(* IEC 61131-3 sources: s32-hmi/, 2 files *)

(* ---- state-machine.st ---- *)
(*
===============================================================================
VOLTAGRID / SEL RTAC MASTER CONTROLLER
STATE-MACHINE SKELETON
Single Master Controller Version
-------------------------------------------------------------------------------
Intent:
- Supervisory coordination only
- Local genset controllers, SEL relays, SEL-2240, OEM controllers retain
  machine/protection ownership
- Master issues permissives, start/stop requests, breaker open/close requests,
  AGC/VCS biases, and orchestrates major sequences
===============================================================================
*)

(*
===============================================================================
TYPE DECLARATIONS
===============================================================================
*)
TYPE E_SYS_STATE :
(
    SYS_INIT := 0,
    SYS_IDLE := 1,
    SYS_NORMAL := 2,
    SYS_PARTY_MODE := 3,
    SYS_BLACKOUT_DETECTED := 4,
    SYS_BLACKOUT_RECOVERY := 5,
    SYS_BLACKSTART_READY := 6,
    SYS_BLACKSTART_ACTIVE := 7,
    SYS_FAULT := 8,
    SYS_ABORTED := 9
);
END_TYPE

TYPE E_SEQ_STATE :
(
    SEQ_IDLE := 0,
    SEQ_START := 1,
    SEQ_CHECK_PERMISSIVES := 2,
    SEQ_ISSUE_COMMAND := 3,
    SEQ_WAIT_FEEDBACK := 4,
    SEQ_VERIFY := 5,
    SEQ_COMPLETE := 6,
    SEQ_FAIL := 7,
    SEQ_ABORT := 8
);
END_TYPE

TYPE E_GEN_MODE :
(
    GEN_BLOCK := 0,
    GEN_STOP := 1,
    GEN_AUTO := 2,
    GEN_MANUAL := 3
);
END_TYPE

TYPE E_GEN_RUN_STATE :
(
    GEN_OFFLINE := 0,
    GEN_STARTING := 1,
    GEN_RUNNING_UNSYNC := 2,
    GEN_SYNCED := 3,
    GEN_STOPPING := 4,
    GEN_TRIPPED := 5,
    GEN_UNAVAILABLE := 6
);
END_TYPE

TYPE E_BREAKER_STATE :
(
    BRK_OPEN := 0,
    BRK_CLOSED := 1,
    BRK_TRANSITION := 2,
    BRK_FAIL := 3,
    BRK_UNKNOWN := 4
);
END_TYPE

TYPE ST_Genset :
STRUCT
    Id                      : INT;
    Enabled                 : BOOL;
    ModeCmd                 : E_GEN_MODE;     (* from HMI *)
    Priority                : INT;            (* 1..100 *)
    EngineHours             : REAL;

    (* permissives / feedback *)
    LocalReadyForDemand     : BOOL;           (* DIA.NE / OEM / Modbus *)
    InAutoAtLocal           : BOOL;
    NoStartBlockAlarms      : BOOL;
    RunningFb               : BOOL;
    SyncCompleteFb          : BOOL;
    GCB_ClosedFb            : BOOL;
    TripFb                  : BOOL;
    DelayedShutdownReqFb    : BOOL;

    (* measured *)
    kW                      : REAL;
    kVAR                    : REAL;
    AvailablekW             : REAL;

    (* supervisory outputs *)
    StartReq                : BOOL;
    StopReq                 : BOOL;
    RemoteBlockCmd          : BOOL;
    PlantEmergencyModeCmd   : BOOL;
    FastDisconnectCmd       : BOOL;
    FullThrottleModeCmd     : BOOL;

    AGC_Enable              : BOOL;
    AGC_Manual              : BOOL;
    AGC_kW_Setpoint         : REAL;
    AGC_kW_Min              : REAL;
    AGC_kW_Max              : REAL;
    AGC_BiasOut             : REAL;           (* abstract bias output *)

    VCS_Enable              : BOOL;
    VCS_Manual              : BOOL;
    VCS_kVAR_Setpoint       : REAL;
    VCS_kVAR_Min            : REAL;
    VCS_kVAR_Max            : REAL;
    VCS_BiasOut             : REAL;           (* abstract bias output *)

    RunState                : E_GEN_RUN_STATE;
    StartPermissive         : BOOL;
    StopPermissive          : BOOL;
    SelectedForStart        : BOOL;
    SelectedForStop         : BOOL;
END_STRUCT
END_TYPE

TYPE ST_Breaker :
STRUCT
    Id                      : INT;
    Name                    : STRING[40];
    ControlEnabled          : BOOL;
    RatedAmps               : INT;

    OpenFb                  : BOOL;
    ClosedFb                : BOOL;
    TripAlarmFb             : BOOL;
    BusVoltage              : REAL;

    OpenCmd                 : BOOL;
    CloseCmd                : BOOL;
    BlockClose              : BOOL;

    State                   : E_BREAKER_STATE;
    SeqState                : E_SEQ_STATE;
END_STRUCT
END_TYPE

TYPE ST_System :
STRUCT
    State                   : E_SYS_STATE;
    PrevState               : E_SYS_STATE;

    HealthyMaster           : BOOL;
    HealthyComms            : BOOL;
    HMI_HeartbeatOk         : BOOL;
    OT_Healthy              : BOOL;

    PartyModeReq            : BOOL;
    PartyModeActive         : BOOL;
    BlackStartEnable        : BOOL;
    BlackStartReq           : BOOL;
    BlackStartActive        : BOOL;

    BlackoutDetected        : BOOL;
    DeadBus34k5             : BOOL;
    DeadBus480              : BOOL;

    IRM_TargetPct           : REAL;
    MinimumSynchronized     : INT;
    MinGensetLoadPct        : REAL;

    Plant_kW_Load           : REAL;
    Plant_kVAR              : REAL;
    MainBus_kV              : REAL;
    MainBus_Hz              : REAL;

    AlarmActive             : BOOL;
    FaultLatched            : BOOL;
    AbortReq                : BOOL;
    ResetReq                : BOOL;
END_STRUCT
END_TYPE

(*
===============================================================================
GLOBAL VARIABLES
===============================================================================
*)
VAR_GLOBAL
    gSys            : ST_System;
    gGensets        : ARRAY[1..46] OF ST_Genset;      (* size adapt per site *)
    gMVBreakers     : ARRAY[1..200] OF ST_Breaker;    (* site-specific *)
    gLVBreakers     : ARRAY[1..200] OF ST_Breaker;    (* site-specific *)
END_VAR

(*
===============================================================================
UTILITY FUNCTIONS
===============================================================================
*)
FUNCTION F_IsDeadBus : BOOL
VAR_INPUT
    Bus_kV          : REAL;
    Nominal_kV      : REAL;
    ThresholdPU     : REAL;       (* e.g. 0.3 *)
END_VAR
F_IsDeadBus := (Bus_kV < (Nominal_kV * ThresholdPU));

FUNCTION F_GensetStartPermissive : BOOL
VAR_INPUT
    Gen             : ST_Genset;
END_VAR
F_GensetStartPermissive :=
    Gen.Enabled
    AND (Gen.ModeCmd = GEN_AUTO)
    AND Gen.LocalReadyForDemand
    AND Gen.InAutoAtLocal
    AND Gen.NoStartBlockAlarms
    AND NOT Gen.TripFb;

FUNCTION F_GensetStopPermissive : BOOL
VAR_INPUT
    Gen             : ST_Genset;
END_VAR
F_GensetStopPermissive :=
    Gen.Enabled
    AND (Gen.RunState = GEN_SYNCED OR Gen.RunState = GEN_RUNNING_UNSYNC)
    AND NOT Gen.TripFb;

FUNCTION F_AverageOnlineLoadPct : REAL
VAR
    i               : INT;
    n               : INT;
    totalPct        : REAL;
    pct             : REAL;
END_VAR
n := 0;
totalPct := 0.0;

FOR i := 1 TO 46 DO
    IF gGensets[i].RunState = GEN_SYNCED THEN
        IF gGensets[i].AvailablekW > 0.0 THEN
            pct := (gGensets[i].kW / gGensets[i].AvailablekW) * 100.0;
            totalPct := totalPct + pct;
            n := n + 1;
        END_IF;
    END_IF;
END_FOR;

IF n > 0 THEN
    F_AverageOnlineLoadPct := totalPct / INT_TO_REAL(n);
ELSE
    F_AverageOnlineLoadPct := 0.0;
END_IF;

FUNCTION F_OnlineGenCount : INT
VAR
    i               : INT;
    n               : INT;
END_VAR
n := 0;
FOR i := 1 TO 46 DO
    IF gGensets[i].RunState = GEN_SYNCED THEN
        n := n + 1;
    END_IF;
END_FOR;
F_OnlineGenCount := n;

FUNCTION F_RequiredGenCountIRM : INT
VAR_INPUT
    PlantLoadkW         : REAL;
    IRM_TargetPct       : REAL;
END_VAR
VAR
    RequiredCapacity    : REAL;
    i                   : INT;
    sortedCap           : ARRAY[1..46] OF REAL;
    sumCap              : REAL;
    cnt                 : INT;
END_VAR

(* Skeleton only:
   Required online count = enough online available kW so that
   reserve margin >= IRM_TargetPct.
*)
RequiredCapacity := PlantLoadkW * (1.0 + (IRM_TargetPct / 100.0));
sumCap := 0.0;
cnt := 0;

FOR i := 1 TO 46 DO
    IF gGensets[i].Enabled THEN
        cnt := cnt + 1;
        sortedCap[cnt] := gGensets[i].AvailablekW;
    END_IF;
END_FOR;

(* TODO: sort by commitment preference / priority class *)
sumCap := 0.0;
F_RequiredGenCountIRM := 0;
FOR i := 1 TO cnt DO
    sumCap := sumCap + sortedCap[i];
    F_RequiredGenCountIRM := F_RequiredGenCountIRM + 1;
    IF sumCap >= RequiredCapacity THEN
        EXIT;
    END_IF;
END_FOR;

(*
===============================================================================
FUNCTION BLOCKS
===============================================================================
*)
FUNCTION_BLOCK FB_GensetState
VAR_INPUT
    Id              : INT;
END_VAR
VAR
    StartPerm       : BOOL;
    StopPerm        : BOOL;
END_VAR

StartPerm := F_GensetStartPermissive(Gen := gGensets[Id]);
StopPerm  := F_GensetStopPermissive(Gen := gGensets[Id]);

gGensets[Id].StartPermissive := StartPerm;
gGensets[Id].StopPermissive  := StopPerm;

IF gGensets[Id].TripFb THEN
    gGensets[Id].RunState := GEN_TRIPPED;

ELSIF gGensets[Id].RunningFb AND gGensets[Id].GCB_ClosedFb AND gGensets[Id].SyncCompleteFb THEN
    gGensets[Id].RunState := GEN_SYNCED;

ELSIF gGensets[Id].RunningFb AND NOT gGensets[Id].GCB_ClosedFb THEN
    gGensets[Id].RunState := GEN_RUNNING_UNSYNC;

ELSIF gGensets[Id].StartReq AND NOT gGensets[Id].RunningFb THEN
    gGensets[Id].RunState := GEN_STARTING;

ELSIF gGensets[Id].StopReq AND gGensets[Id].RunningFb THEN
    gGensets[Id].RunState := GEN_STOPPING;

ELSIF NOT gGensets[Id].RunningFb THEN
    gGensets[Id].RunState := GEN_OFFLINE;

ELSE
    (* hold last *)
END_IF;

FUNCTION_BLOCK FB_AGC_VCS
VAR
    i               : INT;
    OnlineCount     : INT;
    HzError         : REAL;
    kVError         : REAL;
    SharedkWBias    : REAL;
    SharedkVARBias  : REAL;
END_VAR

OnlineCount := F_OnlineGenCount();

(* Skeleton only *)
HzError := 60.0 - gSys.MainBus_Hz;
kVError := 34.5 - gSys.MainBus_kV;

SharedkWBias := HzError * 100.0;
SharedkVARBias := kVError * 100.0;

FOR i := 1 TO 46 DO
    IF gGensets[i].RunState = GEN_SYNCED THEN

        IF gGensets[i].AGC_Enable THEN
            IF gGensets[i].AGC_Manual THEN
                gGensets[i].AGC_BiasOut := gGensets[i].AGC_kW_Setpoint;
            ELSE
                gGensets[i].AGC_BiasOut := SharedkWBias / INT_TO_REAL(MAX(OnlineCount,1));
            END_IF;
        ELSE
            gGensets[i].AGC_BiasOut := 0.0;
        END_IF;

        IF gGensets[i].VCS_Enable THEN
            IF gGensets[i].VCS_Manual THEN
                gGensets[i].VCS_BiasOut := gGensets[i].VCS_kVAR_Setpoint;
            ELSE
                gGensets[i].VCS_BiasOut := SharedkVARBias / INT_TO_REAL(MAX(OnlineCount,1));
            END_IF;
        ELSE
            gGensets[i].VCS_BiasOut := 0.0;
        END_IF;

        (* clamp *)
        IF gGensets[i].AGC_BiasOut < gGensets[i].AGC_kW_Min THEN
            gGensets[i].AGC_BiasOut := gGensets[i].AGC_kW_Min;
        END_IF;
        IF gGensets[i].AGC_BiasOut > gGensets[i].AGC_kW_Max THEN
            gGensets[i].AGC_BiasOut := gGensets[i].AGC_kW_Max;
        END_IF;

        IF gGensets[i].VCS_BiasOut < gGensets[i].VCS_kVAR_Min THEN
            gGensets[i].VCS_BiasOut := gGensets[i].VCS_kVAR_Min;
        END_IF;
        IF gGensets[i].VCS_BiasOut > gGensets[i].VCS_kVAR_Max THEN
            gGensets[i].VCS_BiasOut := gGensets[i].VCS_kVAR_Max;
        END_IF;
    ELSE
        gGensets[i].AGC_BiasOut := 0.0;
        gGensets[i].VCS_BiasOut := 0.0;
    END_IF;
END_FOR;

FUNCTION_BLOCK FB_GMS
VAR
    i                   : INT;
    OnlineCount         : INT;
    RequiredCount       : INT;
    AvgLoadPct          : REAL;
    StartIssued         : INT;
    StopCandidate       : INT;
END_VAR

OnlineCount := F_OnlineGenCount();
RequiredCount := F_RequiredGenCountIRM(
                    PlantLoadkW := gSys.Plant_kW_Load,
                    IRM_TargetPct := gSys.IRM_TargetPct);
IF RequiredCount < gSys.MinimumSynchronized THEN
    RequiredCount := gSys.MinimumSynchronized;
END_IF;

AvgLoadPct := F_AverageOnlineLoadPct();

(* clear selections *)
FOR i := 1 TO 46 DO
    gGensets[i].SelectedForStart := FALSE;
    gGensets[i].SelectedForStop := FALSE;
END_FOR;

(* Party Mode bypasses automatic GMS *)
IF gSys.PartyModeActive THEN
    RETURN;
END_IF;

(* Start logic: IRM has priority *)
IF OnlineCount < RequiredCount THEN
    StartIssued := 0;

    (* Skeleton selection:
       Choose two startable gensets by best priority / least hours tie-break
    *)
    FOR i := 1 TO 46 DO
        IF F_GensetStartPermissive(Gen := gGensets[i]) AND (gGensets[i].RunState = GEN_OFFLINE) THEN
            gGensets[i].SelectedForStart := TRUE;
            gGensets[i].StartReq := TRUE;
            StartIssued := StartIssued + 1;
        END_IF;

        IF StartIssued >= 2 THEN
            EXIT;
        END_IF;
    END_FOR;
END_IF;

(* Stop logic: only if above IRM need and minimum load violated *)
IF (OnlineCount > RequiredCount) AND (AvgLoadPct < gSys.MinGensetLoadPct) THEN
    StopCandidate := 0;

    (* Skeleton selection:
       Highest engine hours among equal priorities, lowest commitment value first
    *)
    FOR i := 1 TO 46 DO
        IF F_GensetStopPermissive(Gen := gGensets[i]) THEN
            StopCandidate := i;
            EXIT;
        END_IF;
    END_FOR;

    IF StopCandidate > 0 THEN
        gGensets[StopCandidate].SelectedForStop := TRUE;
        gGensets[StopCandidate].StopReq := TRUE;
    END_IF;
END_IF;

(* delayed shutdown override *)
FOR i := 1 TO 46 DO
    IF gGensets[i].DelayedShutdownReqFb THEN
        (* maintain IRM by demanding extra gensets *)
        (* skeleton: flag handled naturally by RequiredCount/start logic *)
    END_IF;
END_FOR;

FUNCTION_BLOCK FB_PartyMode
VAR
    i               : INT;
END_VAR

gSys.PartyModeActive := gSys.PartyModeReq;

IF gSys.PartyModeActive THEN
    FOR i := 1 TO 46 DO
        IF F_GensetStartPermissive(Gen := gGensets[i]) THEN
            gGensets[i].StartReq := TRUE;
        END_IF;
    END_FOR;
END_IF;

FUNCTION_BLOCK FB_BlackoutRecovery
VAR
    Seq             : E_SEQ_STATE := SEQ_IDLE;
    TimerExpired    : BOOL;
    i               : INT;
END_VAR

CASE Seq OF

SEQ_IDLE:
    IF gSys.BlackoutDetected THEN
        Seq := SEQ_START;
    END_IF;

SEQ_START:
    (* Verify master and comms healthy *)
    IF gSys.HealthyMaster AND gSys.HealthyComms THEN
        Seq := SEQ_CHECK_PERMISSIVES;
    ELSE
        Seq := SEQ_FAIL;
    END_IF;

SEQ_CHECK_PERMISSIVES:
    gSys.DeadBus34k5 := F_IsDeadBus(Bus_kV := gSys.MainBus_kV, Nominal_kV := 34.5, ThresholdPU := 0.3);
    (* gSys.DeadBus480 to come from LV E-house measurement *)
    IF gSys.DeadBus34k5 AND gSys.DeadBus480 THEN
        Seq := SEQ_ISSUE_COMMAND;
    END_IF;

SEQ_ISSUE_COMMAND:
    (* Open all ICBs + LV feeders required by site logic *)
    FOR i := 1 TO 200 DO
        IF gMVBreakers[i].ControlEnabled THEN
            gMVBreakers[i].OpenCmd := TRUE;
        END_IF;
        IF gLVBreakers[i].ControlEnabled THEN
            gLVBreakers[i].OpenCmd := TRUE;
        END_IF;
    END_FOR;

    (* Start backup diesel through OEM controller / EMCP interface *)
    (* BackupDiesel.StartReq := TRUE; *)
    Seq := SEQ_WAIT_FEEDBACK;

SEQ_WAIT_FEEDBACK:
    (* wait for breaker feedback and backup diesel online *)
    (* skeleton: replace with timers and feedback checks *)
    TimerExpired := FALSE;
    IF NOT TimerExpired THEN
        Seq := SEQ_VERIFY;
    ELSE
        Seq := SEQ_FAIL;
    END_IF;

SEQ_VERIFY:
    (* close critical LV feeders only *)
    (* issue site-specific close list *)
    Seq := SEQ_COMPLETE;

SEQ_COMPLETE:
    gSys.State := SYS_BLACKSTART_READY;
    (* hold complete *)

SEQ_FAIL:
    gSys.AlarmActive := TRUE;
    gSys.FaultLatched := TRUE;
    IF gSys.AbortReq THEN
        Seq := SEQ_ABORT;
    ELSIF gSys.ResetReq THEN
        Seq := SEQ_IDLE;
    END_IF;

SEQ_ABORT:
    gSys.State := SYS_ABORTED;

END_CASE;

FUNCTION_BLOCK FB_BlackStart
VAR
    Seq             : E_SEQ_STATE := SEQ_IDLE;
    i               : INT;
    StartedPrimary  : INT;
END_VAR

CASE Seq OF

SEQ_IDLE:
    IF gSys.BlackStartReq AND gSys.BlackStartEnable AND (gSys.State = SYS_BLACKSTART_READY) THEN
        Seq := SEQ_START;
    END_IF;

SEQ_START:
    gSys.BlackStartActive := TRUE;
    Seq := SEQ_CHECK_PERMISSIVES;

SEQ_CHECK_PERMISSIVES:
    IF gSys.HealthyMaster AND gSys.HealthyComms AND gSys.DeadBus34k5 THEN
        Seq := SEQ_ISSUE_COMMAND;
    ELSE
        Seq := SEQ_FAIL;
    END_IF;

SEQ_ISSUE_COMMAND:
    (* example sequence:
       1) verify all ICBs open
       2) close SYNCON path if required
       3) energize main bus
       4) start/stage gensets
       5) transfer off backup diesel
    *)

    (* step: start two primary gensets *)
    StartedPrimary := 0;
    FOR i := 1 TO 46 DO
        IF F_GensetStartPermissive(Gen := gGensets[i]) THEN
            gGensets[i].StartReq := TRUE;
            StartedPrimary := StartedPrimary + 1;
        END_IF;

        IF StartedPrimary >= 2 THEN
            EXIT;
        END_IF;
    END_FOR;

    Seq := SEQ_WAIT_FEEDBACK;

SEQ_WAIT_FEEDBACK:
    (* wait for running/sync feedback *)
    Seq := SEQ_VERIFY;

SEQ_VERIFY:
    (* if enough primary gensets synced, isolate backup diesel *)
    IF F_OnlineGenCount() >= gSys.MinimumSynchronized THEN
        (* BackupDiesel.StopReq := TRUE; *)
        gSys.BlackStartActive := FALSE;
        Seq := SEQ_COMPLETE;
    ELSE
        Seq := SEQ_FAIL;
    END_IF;

SEQ_COMPLETE:
    gSys.State := SYS_NORMAL;

SEQ_FAIL:
    gSys.AlarmActive := TRUE;
    gSys.FaultLatched := TRUE;
    IF gSys.AbortReq THEN
        Seq := SEQ_ABORT;
    ELSIF gSys.ResetReq THEN
        Seq := SEQ_IDLE;
    END_IF;

SEQ_ABORT:
    gSys.BlackStartActive := FALSE;
    gSys.State := SYS_ABORTED;

END_CASE;

FUNCTION_BLOCK FB_BreakerState
VAR_INPUT
    IsLV            : BOOL;
    Id              : INT;
END_VAR

IF IsLV THEN
    IF gLVBreakers[Id].OpenFb AND NOT gLVBreakers[Id].ClosedFb THEN
        gLVBreakers[Id].State := BRK_OPEN;
    ELSIF gLVBreakers[Id].ClosedFb AND NOT gLVBreakers[Id].OpenFb THEN
        gLVBreakers[Id].State := BRK_CLOSED;
    ELSIF gLVBreakers[Id].TripAlarmFb THEN
        gLVBreakers[Id].State := BRK_FAIL;
    ELSE
        gLVBreakers[Id].State := BRK_UNKNOWN;
    END_IF;
ELSE
    IF gMVBreakers[Id].OpenFb AND NOT gMVBreakers[Id].ClosedFb THEN
        gMVBreakers[Id].State := BRK_OPEN;
    ELSIF gMVBreakers[Id].ClosedFb AND NOT gMVBreakers[Id].OpenFb THEN
        gMVBreakers[Id].State := BRK_CLOSED;
    ELSIF gMVBreakers[Id].TripAlarmFb THEN
        gMVBreakers[Id].State := BRK_FAIL;
    ELSE
        gMVBreakers[Id].State := BRK_UNKNOWN;
    END_IF;
END_IF;

(*
===============================================================================
PROGRAMS
===============================================================================
*)
PROGRAM PRG_InputMapping
VAR
    i               : INT;
END_VAR

(* Map site I/O, FEP tags, relay bits, SEL-2411 data, Modbus data here *)

FOR i := 1 TO 46 DO
    (* Example abstractions only:
       gGensets[i].LocalReadyForDemand := <from SEL-2411 hardwire or Modbus>;
       gGensets[i].RunningFb := <from SEL-2411 or OEM>;
       gGensets[i].GCB_ClosedFb := <from SEL-700G>;
       gGensets[i].SyncCompleteFb := <from OEM / relay>;
       gGensets[i].TripFb := <from OEM/relay>;
       gGensets[i].kW := <analog>;
       gGensets[i].kVAR := <analog>;
       gGensets[i].AvailablekW := <analog>;
       gGensets[i].EngineHours := <Modbus>;
    *)
END_FOR;

(* example Holt-style mapping candidate *)
(*
   Engine Start/Stop write reg: 0x006C
   Engine operating mode read: 0x0000 / 0x00A2
   Starter mode read: 0x021A
   Start-stop state read: 0x009A
   Shutdown active alarm: 0x0281
*)

PROGRAM PRG_SupervisoryState
VAR
    blackoutFB      : FB_BlackoutRecovery;
    blackstartFB    : FB_BlackStart;
END_VAR

gSys.DeadBus34k5 := F_IsDeadBus(Bus_kV := gSys.MainBus_kV, Nominal_kV := 34.5, ThresholdPU := 0.3);

CASE gSys.State OF

SYS_INIT:
    IF gSys.HealthyMaster THEN
        gSys.State := SYS_IDLE;
    END_IF;

SYS_IDLE:
    IF gSys.BlackoutDetected THEN
        gSys.State := SYS_BLACKOUT_DETECTED;
    ELSE
        gSys.State := SYS_NORMAL;
    END_IF;

SYS_NORMAL:
    IF gSys.PartyModeReq THEN
        gSys.State := SYS_PARTY_MODE;
    ELSIF gSys.BlackoutDetected THEN
        gSys.State := SYS_BLACKOUT_DETECTED;
    ELSIF gSys.FaultLatched THEN
        gSys.State := SYS_FAULT;
    END_IF;

SYS_PARTY_MODE:
    IF NOT gSys.PartyModeReq THEN
        gSys.State := SYS_NORMAL;
    END_IF;

SYS_BLACKOUT_DETECTED:
    gSys.State := SYS_BLACKOUT_RECOVERY;

SYS_BLACKOUT_RECOVERY:
    blackoutFB();
    IF gSys.State = SYS_BLACKSTART_READY THEN
        (* transition done in FB *)
    END_IF;

SYS_BLACKSTART_READY:
    IF gSys.BlackStartReq THEN
        gSys.State := SYS_BLACKSTART_ACTIVE;
    END_IF;

SYS_BLACKSTART_ACTIVE:
    blackstartFB();

SYS_FAULT:
    IF gSys.ResetReq THEN
        gSys.FaultLatched := FALSE;
        gSys.State := SYS_IDLE;
    END_IF;

SYS_ABORTED:
    IF gSys.ResetReq THEN
        gSys.State := SYS_IDLE;
    END_IF;

END_CASE;

PROGRAM PRG_GeneratorSupervisor
VAR
    i               : INT;
    genFB           : ARRAY[1..46] OF FB_GensetState;
    agcFB           : FB_AGC_VCS;
    gmsFB           : FB_GMS;
    partyFB         : FB_PartyMode;
END_VAR

FOR i := 1 TO 46 DO
    genFB[i](Id := i);
END_FOR;

partyFB();

IF (gSys.State = SYS_NORMAL) OR (gSys.State = SYS_PARTY_MODE) THEN
    gmsFB();
    agcFB();
END_IF;

PROGRAM PRG_BreakerSupervisor
VAR
    i               : INT;
    mvFB            : ARRAY[1..200] OF FB_BreakerState;
    lvFB            : ARRAY[1..200] OF FB_BreakerState;
END_VAR

FOR i := 1 TO 200 DO
    mvFB[i](IsLV := FALSE, Id := i);
    lvFB[i](IsLV := TRUE, Id := i);
END_FOR;

PROGRAM PRG_OutputMapping
VAR
    i               : INT;
END_VAR

FOR i := 1 TO 46 DO
    (* map supervisory requests to real outputs / comm writes *)

    (* hardwire style *)
    (*
    SEL2411_OUT_Start[i] := PulseFromBool(gGensets[i].StartReq);
    SEL2411_OUT_Stop[i] := PulseFromBool(gGensets[i].StopReq);
    SEL2411_OUT_RemoteBlock[i] := gGensets[i].RemoteBlockCmd;
    SEL2411_AO_kWSetpoint[i] := gGensets[i].AGC_BiasOut;
    SEL2411_AO_kVARSetpoint[i] := gGensets[i].VCS_BiasOut;
    *)

    (* Modbus style alternative *)
    (*
    IF gGensets[i].StartReq THEN
        ModbusWrite(Reg := 16#006C, Value := 2);   (* RUN *)
    ELSIF gGensets[i].StopReq THEN
        ModbusWrite(Reg := 16#006C, Value := 0);   (* STOP *)
    END_IF;
    *)
END_FOR;

FOR i := 1 TO 200 DO
    (* map MV and LV breaker commands to FEP/relay/2240 interface *)
    (* NGVL -> FEP -> GOOSE/MMS/Modbus *)
END_FOR;

PROGRAM PLC_PRG
PRG_InputMapping();
PRG_SupervisoryState();
PRG_GeneratorSupervisor();
PRG_BreakerSupervisor();
PRG_OutputMapping();

(* ---- load-bank-main.st ---- *)
PROGRAM Main_Main_Man
VAR
	Test_Run : BOOL;

	Burn_In : TON;
	Current_Burn_In_Time : TIME;

	Load_Bank_Gateway_Software_Version : DINT;
	Load_Bank_Load_Accept_Sync : DINT;
	Load_Bank_Load_Accept_Reject : DINT;
	Load_Bank_Load_Bank_Count : DINT;
	Load_Bank_Nominal_Voltage : DINT;
	Load_Bank_Nominal_Frequency : DINT;
	Load_Bank_Connection_Mode : DINT;
	Load_Bank_Min_Resistive_Load_Step : UDINT;
	Load_Bank_Measured_Active_Power : DINT;
	Load_Bank_Applied_Resistive_Load : UDINT;
	Load_Bank_Requested_Resistive_Load : UDINT;
	Load_Bank_Requested_Resistive_Load_2 : UDINT;
	Load_Bank_Network_Rescan : DINT;
	Load_Bank_System_Status : DINT;
	Load_Bank_System_Alarms : DINT;
	Load_Bank_Available_Resistive_Load : UDINT;
	Test_Value : DINT;

	Gen_1_kW : UDINT;
	Gen_2_kW : UDINT;
	Gen_3_kW : UDINT;

	Gen_1_52A : BOOL;
	Gen_2_52A : BOOL;
	Gen_3_52A : BOOL;

	Number_of_Gens_Online : UDINT;
	Previous_Number_of_Gens_Online : UDINT;
	Number_of_Gens_Online_Change_Tracker : BOOL;
	Number_of_Gens_Online_Change_Timer : TON;
	New_Gen_Online : BOOL;
	Gen_Shutdown : BOOL;

	// Process variables with default values
    Target_Gen_kW 		: UDINT := 2050;
	Load_Bank_Cap 		: UDINT := 2000; //user limit
	Gen_kW_High_Limit 	: UDINT := 2150;

    // Local variables to receive input from HMI via Modbus write command
    Target_Gen_kW_HMI_Input : UDINT;
	Load_Bank_Cap_HMI_Input : UDINT;
	Gen_kW_High_Limit_HMI_Input : UDINT;

    // Internal flags
    User_SP_Initialized : BOOL := FALSE; // TRUE once user writes at least once
    Last_HMI_SP_Command : UDINT := 0; // Track last valid command

	LB_SP_Initialized : BOOL := FALSE;
	Last_HMI_LB_Command : UDINT := 0;

	kWLimit_SP_Initialized : BOOL := FALSE;
	Last_HMI_kWLimit_Command : UDINT := 0;

	Scaled_Set_Point_To_Measured_Deviation_Cap : DINT;
	Average_Gen_kW : UDINT;
	Gen_kW_Difference : DINT;
	Highest_Gen_kW : UDINT;
	Load_Bank_kW_Set_Point : UDINT;
	Load_Bank_kW_Set_Point_Scaled : UDINT;
	Load_Bank_kW_Set_Point_Byte_1 : UDINT;
	Load_Bank_kW_Set_Point_Byte_2 : UDINT;
	Load_Bank_Step_kW : UDINT;
	Action_Switch : BOOL;

	FirstScan : BOOL := TRUE;

	// Process variable limits
	Target_SP_Min : UDINT := 500;
	Target_SP_Max : UDINT := 2500;

	LB_Min        : UDINT := 500;
    LB_Max        : UDINT; //will be dynamic according to: Load_Bank_Available_Resistive_Load := DINT_TO_UDINT(Modbus_Load_Bank_Available_Resistive_Load.status.stVal); // load bank max capacity div 100 for kw

    kWLimit_Min   : UDINT := 1000;
    kWLimit_Max   : UDINT := 2500;

	// ========== ADDED: AUTO/MANUAL MODE CONTROL VARIABLES ==========
	// Control mode: TRUE = AUTO (automatic control), FALSE = MANUAL (operator-specified setpoint)
	Control_Mode : BOOL := TRUE; // Default to AUTO mode
	Control_Mode_HMI_Input : BOOL;
	Last_HMI_Mode_Command : BOOL := TRUE;
	Mode_Initialized : BOOL := FALSE;

	// Manual mode setpoint and tracking variables
	Manual_Load_Bank_Setpoint : UDINT := 0; // Manual mode setpoint in kW
	Manual_Load_Bank_Setpoint_HMI_Input : UDINT;
	Last_HMI_Manual_SP_Command : UDINT := 0;
	Manual_SP_Initialized : BOOL := FALSE;

	// Manual setpoint limits (dynamic max based on available load bank capacity)
	Manual_SP_Min : UDINT := 0;
	Manual_SP_Max : UDINT; // Will be set to LB_Max dynamically
	// ========== END ADDED VARIABLES ==========

	// ========== ADDED: TEST/LIVE MODE HMI CONTROL VARIABLES ==========
	// Test_Run already declared above: TRUE = Test Mode (no outputs), FALSE = Live Mode (outputs active)
	Test_Mode_HMI_Input : BOOL;
	Last_HMI_Test_Mode_Command : BOOL := TRUE; // Track last command (default TRUE = Test Mode)
	Test_Mode_Initialized : BOOL := FALSE;
	// ========== END ADDED TEST MODE VARIABLES ==========

END_VAR

IF FirstScan THEN
    // Force initial values reconfirmed
	IF NOT User_SP_Initialized AND (Last_HMI_SP_Command = 0) THEN
    	Target_Gen_kW := 2050;
	END_IF;

	IF NOT LB_SP_Initialized AND (Last_HMI_LB_Command = 0) THEN
    	Load_Bank_Cap := 2000;
	END_IF;

	(* Gen_kW_High_Limit default = 2150 *)
	IF NOT kWLimit_SP_Initialized AND (Last_HMI_kWLimit_Command = 0) THEN
    	Gen_kW_High_Limit := 2150;
	END_IF;

	// Clear any stale HMI input
    Target_Gen_kW_HMI_Input := 0;
	Load_Bank_Cap_HMI_Input := 0;
	Gen_kW_High_Limit_HMI_Input := 0;

	// ========== ADDED: Initialize AUTO/MANUAL mode on first scan ==========
	// Default to AUTO mode if not already initialized
	IF NOT Mode_Initialized AND (Last_HMI_Mode_Command = TRUE) THEN
		Control_Mode := TRUE; // Start in AUTO mode
	END_IF;

	// Clear any stale mode and manual setpoint inputs
	Control_Mode_HMI_Input := TRUE;
	Manual_Load_Bank_Setpoint_HMI_Input := 0;
	// ========== END ADDED INITIALIZATION ==========

	// ========== ADDED: Initialize TEST/LIVE mode on first scan ==========
	// Default to TEST mode (Test_Run = TRUE) for safety
	IF NOT Test_Mode_Initialized AND (Last_HMI_Test_Mode_Command = TRUE) THEN
		Test_Run := TRUE; // Start in TEST mode for safety
	END_IF;

	// Clear any stale test mode input
	Test_Mode_HMI_Input := TRUE; // Default to Test Mode
	// ========== END ADDED TEST MODE INITIALIZATION ==========

	Test_Run := 1;

	FirstScan := FALSE;
END_IF

//Initialize the burn in timer
Burn_In();

//Burn in timer used to prevent the
IF NOT Burn_In.IN THEN

	//Test_Run := 0;
	Test_Run := 1;

	//This is the load level, in kW, that the RTAC will try to maintain on each genset
	//Target_Gen_kW := 2050;

	//determines the size of the incremental step changes in the load bank set point.
	//i.e. if the program is increasing the load by 500kW and Load_Bank_Step_kW is set to 50, then the Load Bank Set Point will increase by 50kW during each iteration of the main loop.
	//This incremental increase/decrease will occur roughly once per Cycle Time (as defined in the main controller settings, typically 100 to 500ms)
	//Cycle Time is 100ms as of 25 SEP 25
	Load_Bank_Step_kW := 50;

	//Load_Bank_Cap := 2000;
	//Gen_kW_High_Limit := 2150;
	Scaled_Set_Point_To_Measured_Deviation_Cap := 10000;

	Burn_In.PT := T#30S;
	Burn_In.IN := 1;
	Modbus_Load_Bank_Load_Accept_Sync.oper.ctlVal := 0;
	Modbus_Load_Bank_Load_Accept_Sync.oper.trigger := 1;
END_IF

//Just here to show the current burn in time after going online in the AcSELerator RTAC software
Current_Burn_In_Time := Burn_In.ET;

//Main IF Loop - data is loaded into variables for use by the main algorithm, the difference between the average genset load and the target genset load is calculated, then the load bank set point is updated.
IF TRUE THEN

	// User input modbus write commands (HMI -> RTAC)
	HMI_Modbus_Server_Tags_Target_kW_Input.oper.trigger := NOT HMI_Modbus_Server_Tags_Target_kW_Input.oper.trigger;
	Target_Gen_kW_HMI_Input := DINT_TO_UDINT(HMI_Modbus_Server_Tags_Target_kW_Input.oper.ctlVal);
	HMI_Modbus_Server_Tags_Load_Bank_Cap_Input.oper.trigger := NOT HMI_Modbus_Server_Tags_Load_Bank_Cap_Input.oper.trigger;
	Load_Bank_Cap_HMI_Input := DINT_TO_UDINT(HMI_Modbus_Server_Tags_Load_Bank_Cap_Input.oper.ctlVal);
	HMI_Modbus_Server_Tags_kW_High_Limit_Input.oper.trigger := NOT HMI_Modbus_Server_Tags_kW_High_Limit_Input.oper.trigger;
	Gen_kW_High_Limit_HMI_Input := DINT_TO_UDINT(HMI_Modbus_Server_Tags_kW_High_Limit_Input.oper.ctlVal);

	// Detect new HMI command
	IF Target_Gen_kW_HMI_Input <> Last_HMI_SP_Command THEN

		IF Target_Gen_kW_HMI_Input < Target_SP_Min THEN
			Target_Gen_kW := Target_SP_Min;
		ELSIF Target_Gen_kW_HMI_Input > Target_SP_Max THEN
			Target_Gen_kW := Target_SP_Max;
		ELSE
			Target_Gen_kW := Target_Gen_kW_HMI_Input;
		END_IF;

		User_SP_Initialized := TRUE;
		Last_HMI_SP_Command := Target_Gen_kW_HMI_Input;
	END_IF;

	// HMI feedback target load set point (RTAC → HMI)
	HMI_Modbus_Server_Tags_Target_kW.status.stVal := UDINT_TO_DINT(Target_Gen_kW);
	HMI_Modbus_Server_Tags_Target_kW.oper.trigger := NOT HMI_Modbus_Server_Tags_Target_kW.oper.trigger;

	// Detect new load bank cap command from HMI
	IF Load_Bank_Cap_HMI_Input <> Last_HMI_LB_Command THEN

		IF Load_Bank_Cap_HMI_Input < LB_Min THEN
			Load_Bank_Cap := LB_Min;
		ELSIF Load_Bank_Cap_HMI_Input > LB_Max THEN
			Load_Bank_Cap := LB_Max;
		ELSE
			Load_Bank_Cap := Load_Bank_Cap_HMI_Input;
		END_IF;

		LB_SP_Initialized := TRUE;
		Last_HMI_LB_Command := Load_Bank_Cap_HMI_Input;
	END_IF;

	// HMI load bank cap feedback (RTAC → HMI)
	HMI_Modbus_Server_Tags_Load_Bank_Cap.status.stVal := UDINT_TO_DINT(Load_Bank_Cap);
	HMI_Modbus_Server_Tags_Load_Bank_Cap.oper.trigger := NOT HMI_Modbus_Server_Tags_Load_Bank_Cap.oper.trigger;

	// Detect new kW high limit command from HMI
	IF Gen_kW_High_Limit_HMI_Input <> Last_HMI_kWLimit_Command THEN

		IF Gen_kW_High_Limit_HMI_Input < kWLimit_Min THEN
			Gen_kW_High_Limit := kWLimit_Min;
		ELSIF Gen_kW_High_Limit_HMI_Input > kWLimit_Max THEN
			Gen_kW_High_Limit := kWLimit_Max;
		ELSE
			Gen_kW_High_Limit := Gen_kW_High_Limit_HMI_Input;
		END_IF;

		kWLimit_SP_Initialized := TRUE;
		Last_HMI_kWLimit_Command := Gen_kW_High_Limit_HMI_Input;
	END_IF;

	// HMI kW high limit feedback (RTAC → HMI)
	HMI_Modbus_Server_Tags_kW_High_Limit.status.stVal := UDINT_TO_DINT(Gen_kW_High_Limit);
	HMI_Modbus_Server_Tags_kW_High_Limit.oper.trigger := NOT HMI_Modbus_Server_Tags_kW_High_Limit.oper.trigger;

	// ========== ADDED: AUTO/MANUAL MODE HMI INTERFACE ==========
	// Read control mode selection from HMI (TRUE = AUTO, FALSE = MANUAL)
	HMI_Modbus_Server_Tags_Control_Mode_Input.oper.trigger := NOT HMI_Modbus_Server_Tags_Control_Mode_Input.oper.trigger;
	Control_Mode_HMI_Input := HMI_Modbus_Server_Tags_Control_Mode_Input.oper.ctlVal <> 0; // Convert DINT to BOOL (0=FALSE/MANUAL, 1=TRUE/AUTO)

	// Detect mode change command from HMI
	IF Control_Mode_HMI_Input <> Last_HMI_Mode_Command THEN
		Control_Mode := Control_Mode_HMI_Input;
		Mode_Initialized := TRUE;
		Last_HMI_Mode_Command := Control_Mode_HMI_Input;

		// When switching to MANUAL mode, initialize manual setpoint with current auto setpoint (bumpless transfer)
		IF NOT Control_Mode THEN
			Manual_Load_Bank_Setpoint := Load_Bank_kW_Set_Point;
		END_IF;
	END_IF;

	// Send control mode feedback to HMI (RTAC → HMI)
	HMI_Modbus_Server_Tags_Control_Mode.status.stVal := BOOL_TO_DINT(Control_Mode); // Convert BOOL to DINT (TRUE=1/AUTO, FALSE=0/MANUAL)
	HMI_Modbus_Server_Tags_Control_Mode.oper.trigger := NOT HMI_Modbus_Server_Tags_Control_Mode.oper.trigger;

	// Read manual load bank setpoint from HMI
	HMI_Modbus_Server_Tags_Manual_Load_Bank_SP_Input.oper.trigger := NOT HMI_Modbus_Server_Tags_Manual_Load_Bank_SP_Input.oper.trigger;
	Manual_Load_Bank_Setpoint_HMI_Input := DINT_TO_UDINT(HMI_Modbus_Server_Tags_Manual_Load_Bank_SP_Input.oper.ctlVal);

	// Update dynamic maximum limit for manual setpoint (based on available load bank capacity)
	Manual_SP_Max := LB_Max;

	// Detect new manual setpoint command from HMI
	IF Manual_Load_Bank_Setpoint_HMI_Input <> Last_HMI_Manual_SP_Command THEN

		// Apply min/max limits to manual setpoint
		IF Manual_Load_Bank_Setpoint_HMI_Input < Manual_SP_Min THEN
			Manual_Load_Bank_Setpoint := Manual_SP_Min;
		ELSIF Manual_Load_Bank_Setpoint_HMI_Input > Manual_SP_Max THEN
			Manual_Load_Bank_Setpoint := Manual_SP_Max;
		ELSE
			Manual_Load_Bank_Setpoint := Manual_Load_Bank_Setpoint_HMI_Input;
		END_IF;

		Manual_SP_Initialized := TRUE;
		Last_HMI_Manual_SP_Command := Manual_Load_Bank_Setpoint_HMI_Input;
	END_IF;

	// Send manual setpoint feedback to HMI (RTAC → HMI)
	HMI_Modbus_Server_Tags_Manual_Load_Bank_SP.status.stVal := UDINT_TO_DINT(Manual_Load_Bank_Setpoint);
	HMI_Modbus_Server_Tags_Manual_Load_Bank_SP.oper.trigger := NOT HMI_Modbus_Server_Tags_Manual_Load_Bank_SP.oper.trigger;
	// ========== END ADDED AUTO/MANUAL MODE HMI INTERFACE ==========

	// ========== ADDED: TEST/LIVE MODE HMI INTERFACE ==========
	// Read test mode selection from HMI (TRUE = Test Mode, FALSE = Live Mode)
	// Register 17: Test_Mode_Input (HMI → RTAC)
	HMI_Modbus_Server_Tags_Test_Mode_Input.oper.trigger := NOT HMI_Modbus_Server_Tags_Test_Mode_Input.oper.trigger;
	Test_Mode_HMI_Input := HMI_Modbus_Server_Tags_Test_Mode_Input.oper.ctlVal <> 0; // Convert DINT to BOOL (0=FALSE/Live, 1=TRUE/Test)

	// Detect test mode change command from HMI
	IF Test_Mode_HMI_Input <> Last_HMI_Test_Mode_Command THEN
		Test_Run := Test_Mode_HMI_Input; // TRUE = Test Mode (outputs disabled), FALSE = Live Mode (outputs enabled)
		Test_Mode_Initialized := TRUE;
		Last_HMI_Test_Mode_Command := Test_Mode_HMI_Input;
	END_IF;

	// Send test mode feedback to HMI (RTAC → HMI)
	// Register 16: Test_Mode (RTAC → HMI)
	HMI_Modbus_Server_Tags_Test_Mode.status.stVal := BOOL_TO_DINT(Test_Run); // Convert BOOL to DINT (TRUE=1/Test, FALSE=0/Live)
	HMI_Modbus_Server_Tags_Test_Mode.oper.trigger := NOT HMI_Modbus_Server_Tags_Test_Mode.oper.trigger;
	// ========== END ADDED TEST/LIVE MODE HMI INTERFACE ==========

	//Real-Time Modbus data from the Load Bank Gateway is loaded into internal variables
	Load_Bank_Gateway_Software_Version := Modbus_Load_Bank_Gateway_Software_Version.status.stVal;
	Load_Bank_Load_Accept_Sync := Modbus_Load_Bank_Load_Accept_Sync.status.stVal;
	Load_Bank_Requested_Resistive_Load := DINT_TO_UDINT(Modbus_Load_Bank_Requested_Resistive_Load.status.stVal);
	Load_Bank_Load_Accept_Reject := Modbus_Load_Bank_Load_Accept_Reject.status.stVal;
	Load_Bank_Load_Bank_Count := Modbus_Load_Bank_Load_Bank_Count.status.stVal;
	Load_Bank_Nominal_Voltage := Modbus_Load_Bank_Nominal_Voltage.status.stVal;
	Load_Bank_Nominal_Frequency := Modbus_Load_Bank_Nominal_Frequency.status.stVal;
	Load_Bank_Connection_Mode := Modbus_Load_Bank_Connection_Mode.status.stVal;
	Load_Bank_Min_Resistive_Load_Step := DINT_TO_UDINT(Modbus_Load_Bank_Min_Resistive_Load_Step.status.stVal);
	Load_Bank_Measured_Active_Power := Modbus_Load_Bank_Measured_Active_Power.status.stVal;
	Load_Bank_Applied_Resistive_Load := DINT_TO_UDINT(Modbus_Load_Bank_Applied_Resistive_Load.status.stVal);
	Load_Bank_System_Status := Modbus_Load_Bank_System_Status.status.stVal;
	Load_Bank_System_Alarms := Modbus_Load_Bank_System_Alarms.status.stVal;
	Load_Bank_Available_Resistive_Load := DINT_TO_UDINT(Modbus_Load_Bank_Available_Resistive_Load.status.stVal); // load bank max capacity div 100 for kw

	// Calculate the Maximum kW limit by removing the scaling factor
	// Ensure we don't divide by zero if the load bank is offline (though 0/100 is just 0)
	LB_Max := Load_Bank_Available_Resistive_Load / 100;

	IF Load_Bank_Load_Accept_Sync = 1 AND Burn_in.Q THEN
		Modbus_Load_Bank_Load_Accept_Sync.oper.ctlVal := 0;
		Modbus_Load_Bank_Load_Accept_Sync.oper.trigger := NOT Modbus_Load_Bank_Load_Accept_Sync.oper.trigger;
	END_IF

	//Real-Time Three-phase power measurement from each generator is loaded into an internal variable
	Gen_1_kW := REAL_TO_UDINT(SEL_700G_1_SEL.FM_INST_P3X.mag / 1000);
	Gen_2_kW := REAL_TO_UDINT(SEL_700G_2_SEL.FM_INST_P3X.mag / 1000);
	Gen_3_kW := REAL_TO_UDINT(SEL_700G_3_SEL.FM_INST_P3X.mag / 1000);

	//Serve up genset KW to HMI via modbus tcp slave
	HMI_Modbus_Server_Tags_Kw_GenSet_1.stVal := UDINT_TO_DINT(Gen_1_kW);
	HMI_Modbus_Server_Tags_Kw_GenSet_2.stVal := UDINT_TO_DINT(Gen_2_kW);
	HMI_Modbus_Server_Tags_Kw_GenSet_3.stVal := UDINT_TO_DINT(Gen_3_kW);

	//Real-Time GCB breaker-closed status from each generator is loaded into an internal variable
	Gen_1_52A := SEL_700G_1_SEL.FM_INST_52AX.stVal;
	Gen_2_52A := SEL_700G_2_SEL.FM_INST_52AX.stVal;
	Gen_3_52A := SEL_700G_3_SEL.FM_INST_52AX.stVal;

	//Serve up circuit breaker status to HMI
	HMI_Modbus_Server_Tags_52A_Status_GenSet_1.status.stVal := Gen_1_52A;
	HMI_Modbus_Server_Tags_52A_Status_GenSet_2.status.stVal := Gen_2_52A;
	HMI_Modbus_Server_Tags_52A_Status_GenSet_3.status.stVal := Gen_3_52A;

	//Generator breaker statuses are used to determine how many generators are synchronized and closed into the bus
	Number_of_Gens_Online := BOOL_TO_UDINT(Gen_1_52A) + BOOL_TO_UDINT(Gen_2_52A) + BOOL_TO_UDINT(Gen_3_52A);

	//Average generator load is calculated by dividing the sum of all genset loads by the number of gensets online
	IF Number_of_Gens_Online > 0 THEN
			Average_Gen_kW := (Gen_1_kW + Gen_2_kW + Gen_3_kW) / Number_of_Gens_Online;
	ELSE
		Average_Gen_kW := 0;
	END_IF

	//The differnce between the
	IF Average_Gen_kW > 0 THEN
		Gen_kW_Difference := UDINT_TO_DINT(Target_Gen_kW) - UDINT_TO_DINT(Average_Gen_kW);
	ELSE
		Gen_kW_Difference := 0;
	END_IF

	//The highest individual generator load is determined so that load bank load increases can be prevented if there is risk of overloading a unit
	Highest_Gen_kW := MAX(Gen_1_kW, Gen_2_kW, Gen_3_kW);

	// ========== MODIFIED: Wrapped control logic with AUTO/MANUAL mode selection ==========
	IF Control_Mode THEN
		// ===== AUTO MODE - Automatic control algorithm (original logic) =====
		IF ((Load_Bank_kW_Set_Point_Scaled) <= DINT_TO_UDINT(Load_Bank_Measured_Active_Power + Scaled_Set_Point_To_Measured_Deviation_Cap)) AND NOT Modbus_Load_Bank_Requested_Resistive_Load.oper.trigger THEN
			//The Load Bank Set Point is increased, decreased, or remains the same depending on the average generator load (in order to maintain the gensets at target load)
			IF Highest_Gen_kW >= Gen_kW_High_Limit AND Load_Bank_kW_Set_Point >= 200 THEN
				Load_Bank_kW_Set_Point := Load_Bank_kW_Set_Point - (Load_Bank_Step_kW * 2);
			ELSE
				IF Gen_kW_Difference <= (-1 * UDINT_TO_DINT(Load_Bank_Step_kW)) AND Load_Bank_kW_Set_Point >= 100 THEN
					Load_Bank_kW_Set_Point := Load_Bank_kW_Set_Point - (Load_Bank_Step_kW);
				ELSE
					IF Gen_kW_Difference > UDINT_TO_DINT(Load_Bank_Step_kW) AND Highest_Gen_kW <= Gen_kW_High_Limit AND Load_Bank_kW_Set_Point <= Load_Bank_Cap THEN
						Load_Bank_kW_Set_Point := Load_Bank_kW_Set_Point + Load_Bank_Step_kW;
					ELSE
						IF Load_Bank_kW_Set_Point_Scaled > DINT_TO_UDINT(Load_Bank_Measured_Active_Power + Scaled_Set_Point_To_Measured_Deviation_Cap) THEN
							Load_Bank_kW_Set_Point := Load_Bank_kW_Set_Point - Load_Bank_Step_kW * 2;
						END_IF
					END_IF
				END_IF
			END_IF
		ELSE
			IF((Load_Bank_kW_Set_Point_Scaled) >= DINT_TO_UDINT(Load_Bank_Measured_Active_Power + Scaled_Set_Point_To_Measured_Deviation_Cap + 10000)) THEN
				Load_Bank_kW_Set_Point := Load_Bank_kW_Set_Point - Load_Bank_Step_kW * 2;
			END_IF
		END_IF
	ELSE
		// ===== MANUAL MODE - Operator-specified setpoint (no automatic control) =====
		// In manual mode, the load bank setpoint is directly set by the operator via HMI
		// The automatic control algorithm is bypassed
		Load_Bank_kW_Set_Point := Manual_Load_Bank_Setpoint;
	END_IF;
	// ========== END MODIFIED CONTROL LOGIC ==========

	// Scales the Load_Bank_kW_Set_Point value so it can be written to the load bank gateway modbus register
	Load_Bank_kW_Set_Point_Scaled := Load_Bank_kW_Set_Point * 100;

	//Modbus Holding Registers are loaded with the values required for the load bank(s) to increase/decrease to the new desired load level
	Modbus_Load_Bank_Requested_Resistive_Load.oper.ctlVal := UDINT_TO_DINT(Load_Bank_kW_Set_Point_Scaled);

END_IF

	//If the code isn't in test mode, the new Modbus Holding Register values are sent to the Load Bank Gateway
	//This is the control action which should result in a change in load bank load levels if required
IF Test_Run = 0 AND Burn_In.Q THEN
	Modbus_Load_Bank_Requested_Resistive_Load.oper.trigger := NOT Modbus_Load_Bank_Requested_Resistive_Load.oper.trigger;
	//Modbus_Load_Bank_Requested_Resistive_Load_2.oper.trigger := NOT Modbus_Load_Bank_Requested_Resistive_Load_2.oper.trigger;
	//Modbus_Load_Bank_Load_Accept_Reject.oper.trigger := NOT Modbus_Load_Bank_Load_Accept_Reject.oper.trigger;
END_IF
